// TwinCAT 3 PLC project PLCProject
// ProgramVersion: 3.1.4023.0
// libraries:
//   Tc2_Standard, * (Beckhoff Automation GmbH)
//   Tc2_System, * (Beckhoff Automation GmbH)
//   Tc3_Module, * (Beckhoff Automation GmbH)
// project tree:
//   / PlcTask.TcTTO
//   POUs/ MAIN.TcPOU
// real-time tasks:
//   TASK PlcTask: cycle T#1ms, priority 20, ADS port 350
// motion (NC):
//   TASK NC-Task 1 SAF: cycle T#2ms, priority 4, ADS port 501
//   TASK NC-Task 1 SVB: cycle T#10ms, priority 8, ADS port 511
//   AXIS Axis 1 (id 1)
//     OtherSettings: AllowMotionCmdToSlave=true
//     encoder EncType=19
//       EncPara: MaxCount=#xffffffff
//     drive DrvType=16
//       DrvPara: MaxCount=#xffffffff
//         Analog: TorqueSetpointScale=10, ScaleFactorActTorque=0.1
//         TimeComp: TaskDelayCycles=1
//     controller CtrType=1
//       CtrPara: PriorControlFactor=1
//         Observer: BandWidth=20
// I/O:
//   DEVICE Device 1 (EtherCAT), AmsNetId 192.168.212.233.2.1
//     Box 3 (AXL F BK EC) [AXL F BK EC, Axioline EtherCAT Fieldbus coupler]
//       modules: Module 1 (AXL F DI16/4 2F), Module 2 (AXL F DI16/4 2F), Module 3 (AXL F DI16/4 2F), Module 4 (AXL F DO8/2 2A 1H), Module 5 (AXL F DO8/2 2A 1H), Module 6 (AXL F DO8/2 2A 1H), Module 7 (AXL F AI8 1F), Module 8 (AXL F AI8 1F), Module 9 (AXL F AI8 1F), Module 10 (AXL F AI8 1F), Module 11 (AXL F AO8 1F), Module 12 (AXL F RTD4 1H), Module 13 (AXL F RTD4 1H), Module 14 (AXL F RTD4 1H), Module 15 (AXL F RTD4 1H)
//     Box 5 (AXL F BK EC) [AXL F BK EC, Axioline EtherCAT Fieldbus coupler]
//       modules: Module 1 (AXL F DI16/4 2F), Module 2 (AXL F DOR4/2 AC/220DC 1F), Module 3 (AXL F AI8 1F), Module 4 (AXL F AI8 1F), Module 5 (AXL F AI8 1F)
//     Drive 6 (Ax Series) [Ax Series]
//     Box 8 (AXL F BK EC) [AXL F BK EC, Axioline EtherCAT Fieldbus coupler]
//       modules: Module 1 (AXL F DI16/4 2F), Module 2 (AXL F DI16/4 2F), Module 3 (AXL F DI16/4 2F), Module 4 (AXL F DI16/4 2F), Module 5 (AXL F DOR4/2 AC/220DC 1F), Module 6 (AXL F AI8 1F), Module 7 (AXL F AI8 1F), Module 8 (AXL F AI8 1F)
//     Box 9 (AXL F BK EC) [AXL F BK EC, Axioline EtherCAT Fieldbus coupler]
//       modules: Module 1 (AXL F AO8 1F), Module 2 (AXL F RTD4 1H), Module 3 (AXL F RTD4 1H), Module 4 (AXL F RTD4 1H), Module 5 (AXL F RTD4 1H)
//     Box 10 (AXL F BK EC) [AXL F BK EC, Axioline EtherCAT Fieldbus coupler]
//       modules: Module 1 (AXL F DI16/4 2F), Module 2 (AXL F DOR4/2 AC/220DC 1F), Module 3 (AXL F AI8 1F)
//     Box 11 (AXL F BK EC) [AXL F BK EC, Axioline EtherCAT Fieldbus coupler]
//       modules: Module 1 (AXL F DI16/4 2F), Module 2 (AXL F DOR4/2 AC/220DC 1F), Module 3 (AXL F AI8 1F)
// variable links:
//   PLCProject/PLCProject Instance <-> Device 1 (EtherCAT)/Box 3 (AXL F BK EC)
//     PlcTask Inputs/MAIN.bVariableToLink <-> Module 1 (AXL F DI16/4 2F)/Digital Input Channels/DI Channel 01 (Terminal Point 00)

CONFIGURATION PLCProject
    RESOURCE PLC ON TwinCAT3
        TASK PlcTask(INTERVAL := T#1ms, PRIORITY := 20);
        PROGRAM MAIN WITH PlcTask : MAIN;
    END_RESOURCE
END_CONFIGURATION

// ---- POUs/MAIN.TcPOU
PROGRAM MAIN
VAR
	bVariableToLink  AT %I* : BOOL;
	
END_VAR

END_PROGRAM
